// TIA Portal V17 export
// export: Created 2022-07-20T07:01:31.8354759Z, ExportSetting WithDefaults, DisplayName Totally Integrated Automation Portal, DisplayVersion V17, DisplayName TIA Portal Openness, DisplayVersion V17, DisplayName TIA Portal Version Control Interface, DisplayVersion V17, DisplayName SINAMICS Startdrive Advanced, DisplayVersion V17, DisplayName SINAMICS Startdrive G130, G150, S120, S150, SINAMICS MV, S210, DisplayVersion V17, DisplayName SINAMICS Startdrive G110M, G120, G120C, G120D, G120P, G115D, DisplayVersion V17, DisplayName STEP 7 Professional, DisplayVersion V17, DisplayName STEP 7 Safety, DisplayVersion V17, DisplayName WinCC Advanced, DisplayVersion V17
FUNCTION "FC10332_DWordTo2Words" : Void   // FC10032, LAD
TITLE = FC10011_DintTo2Int
{ S7_Optimized_Access := 'TRUE' }
AUTHOR : Anirouddh
FAMILY : 1001x_CONVERT
VERSION : 1.0
// Release note : 
// 1.0 - Feature developped
// stored: AutoNumber false, IsIECCheckEnabled false, SetENOAutomatically false, UDAEnableTagReadback false
   VAR_INPUT
      DWord_Input : DWord;
   END_VAR
   VAR_OUTPUT
      Word_HighWeight : Word;
      Word_LowWeight : Word;
   END_VAR
BEGIN

REGION Network 1 (SCL)
   #Word_LowWeight.%X0 := #DWord_Input.%X0;
   #Word_LowWeight.%X1 := #DWord_Input.%X1;
   #Word_LowWeight.%X2 := #DWord_Input.%X2;
   #Word_LowWeight.%X3 := #DWord_Input.%X3;
   #Word_LowWeight.%X4 := #DWord_Input.%X4;
   #Word_LowWeight.%X5 := #DWord_Input.%X5;
   #Word_LowWeight.%X6 := #DWord_Input.%X6;
   #Word_LowWeight.%X7 := #DWord_Input.%X7;
   #Word_LowWeight.%X8 := #DWord_Input.%X8;
   #Word_LowWeight.%X9 := #DWord_Input.%X9;
   #Word_LowWeight.%X10 := #DWord_Input.%X10;
   #Word_LowWeight.%X11 := #DWord_Input.%X11;
   #Word_LowWeight.%X12 := #DWord_Input.%X12;
   #Word_LowWeight.%X13 := #DWord_Input.%X13;
   #Word_LowWeight.%X14 := #DWord_Input.%X14;
   #Word_LowWeight.%X15 := #DWord_Input.%X15;

   #Word_HighWeight.%X0 := #DWord_Input.%X16;
   #Word_HighWeight.%X1 := #DWord_Input.%X17;
   #Word_HighWeight.%X2 := #DWord_Input.%X18;
   #Word_HighWeight.%X3 := #DWord_Input.%X19;
   #Word_HighWeight.%X4 := #DWord_Input.%X20;
   #Word_HighWeight.%X5 := #DWord_Input.%X21;
   #Word_HighWeight.%X6 := #DWord_Input.%X22;
   #Word_HighWeight.%X7 := #DWord_Input.%X23;
   #Word_HighWeight.%X8 := #DWord_Input.%X24;
   #Word_HighWeight.%X9 := #DWord_Input.%X25;
   #Word_HighWeight.%X10 := #DWord_Input.%X26;
   #Word_HighWeight.%X11 := #DWord_Input.%X27;
   #Word_HighWeight.%X12 := #DWord_Input.%X28;
   #Word_HighWeight.%X13 := #DWord_Input.%X29;
   #Word_HighWeight.%X14 := #DWord_Input.%X30;
   #Word_HighWeight.%X15 := #DWord_Input.%X31;
END_REGION
END_FUNCTION
